// SIMATIC STEP 7 (V5.x) project PROJECT-ETHERNET_en
// CPU: CPU 414-2 DP(1)
// CPU: CPU 414-2 DP(1)
// CPU: CPU 414-2 DP(1)
// station: P_ADR_BUS
// station: Hardware
// station: SIMATIC 400(3)
// station: P_ADR_BUS
// station: Hardware
// station: SIMATIC 400(2)
// station: P_ADR_BUS
// station: Hardware
// station: SIMATIC 400(1)
// program: S7 Program(1)
// program: S7 Program(1)
// program: S7 Program(1)

SYMBOL_TABLE
"AG_SEND"	FC 5	FC 5	// AG SEND
"AG_RECV"	FC 6	FC 6	// AG RECEIVE
END_SYMBOL_TABLE

// FC 5: know-how protected block, not included

// FC 6: know-how protected block, not included

FUNCTION FC 29 : VOID
VERSION : 0.1
BEGIN
NETWORK
TITLE =
      A     T 4;	//time downwards
      JC    runt;
st_1: A     M 40.1;	//start timer 3
      L     S5T#3S;	//LED upwards 3 sec
      SE    T 3;
      A     T 3;
      R     M 40.1;
      JC    hoch;	//jump for upwards
      AN    T 3;
      S     M 40.1;
      S     M 40.2;
runt: A     M 40.2;	//start timer 4
      L     S5T#3S;	//LED downwards 3 sec
      SE    T 4;
      A     T 4;
      R     M 40.2;
      AN    T 4;
      S     M 40.2;
      JC    st_1;
      A     M 40.0;
      L     S5T#100MS;
      SE    T 1;
      A     T 1;
      R     M 40.0;
      A     T 1;
      JC    weit;
      AN    T 1;
      S     M 40.0;
      L     MW 70;
      L     0;
      <>D;
      JC    los1;
      TAK;
      +     1;
      T     MW 70;
      T     DB30.DBW 1;
      BEU;
los1: L     MW 70;
      L     2;
      *D;
      T     MW 70;
      T     DB30.DBW 1;
      L     L#32768;
      <>D;
      BEC;
      L     0;
      T     MW 70;
weit: BEU;
hoch: A     M 40.3;
      L     S5T#100MS;
      SE    T 1;
      A     T 1;
      R     M 40.3;
      A     T 1;
      JC    weit;
      AN    T 1;
      S     M 40.3;
      L     MW 70;
      L     0;
      <>D;
      JC    los2;
      TAK;
      +     L#32768;
      T     MW 70;
      T     DB30.DBW 1;
      BEU;
los2: L     MW 70;
      L     2;
      /D;
      T     MW 70;
      T     DB30.DBW 1;
      L     1;
      <>D;
      BEC;
      L     0;
      T     MW 70;
      BE;
END_FUNCTION

FUNCTION FC 30 : VOID
TITLE = send
//SIMATIC 400 Station 1
//
//Sends data via ISO transport connection with ID=1.
//Starting at byte 1 in DB30, 4 bytes are going to be send.
//
VERSION : 0.0
BEGIN
NETWORK
TITLE =
      O     M 50.0;
      ON    M 50.0;
      S     M 50.0;
      CALL  "AG_SEND" (
           $1                       := P#M 50.0,
           $2                       := 1,
           $3                       := 512,
           $4                       := P#DB30.DBX 1.0 BYTE 240,
           $5                       := 4,
           $6                       := M 1.2,
           $7                       := M 1.3,
           $8                       := P#M 200.0);	//AG_SEND
      BE;
END_FUNCTION

FUNCTION FC 31 : VOID
TITLE = receive
//SIMATIC 400 Station 1
//
//Receives data via ISO transport connection with ID=1.
//Data are accepted in DB31, starting at byte 1.
VERSION : 0.0
BEGIN
NETWORK
TITLE =
      CALL  "AG_RECV" (
           $1                       := 1,
           $2                       := 512,
           $3                       := P#DB31.DBX 1.0 BYTE 240,
           $4                       := P#M 1.0,
           $5                       := M 1.1,
           $6                       := P#M 202.0,
           $7                       := P#M 10.0);	//AG_RECV
      L     DB31.DBW 1;
      T     QW 0;
      BE;
END_FUNCTION

ORGANIZATION_BLOCK OB 1
//Station 1
VERSION : 0.1
VAR_TEMP
  OB1_EV_CLASS : BYTE ;	//Bits 0-3 = 1 (Coming event), Bits 4-7 = 1 (Event class 1)
  OB1_SCAN_1 : BYTE ;	//1 (Cold restart scan 1 of OB 1), 3 (Scan 2-n of OB 1)
  OB1_PRIORITY : BYTE ;	//1 (Priority of 1 is lowest)
  OB1_OB_NUMBR : BYTE ;	//1 (Organization block 1, OB1)
  OB1_RESERVED_1 : BYTE ;	//Reserved for system
  OB1_RESERVED_2 : BYTE ;	//Reserved for system
  OB1_PREV_CYCLE : INT ;	//Cycle time of previous OB1 scan (milliseconds)
  OB1_MIN_CYCLE : INT ;	//Minimum cycle time of OB1 (milliseconds)
  OB1_MAX_CYCLE : INT ;	//Maximum cycle time of OB1 (milliseconds)
  OB1_DATE_TIME : DATE_AND_TIME ;	//Date and time OB1 started
END_VAR
BEGIN
NETWORK
TITLE =
      CALL  FC 29;
      CALL  FC 30;
      CALL  FC 31;
      BE;
END_ORGANIZATION_BLOCK

ORGANIZATION_BLOCK OB 100
TITLE = Start up
//Station1
VERSION : 0.0
VAR_TEMP
  OB100_EV_CLASS : BYTE ;	//16#13, Event class 1, Entering event state, Event logged in diagnostic buffer
  OB100_STRTUP : BYTE ;	//16#81/82/83/84 Method of startup
  OB100_PRIORITY : BYTE ;	//27 (Priority of 1 is lowest)
  OB100_OB_NUMBR : BYTE ;	//100 (Organization block 100, OB100)
  OB100_RESERVED_1 : BYTE ;	//Reserved for system
  OB100_RESERVED_2 : BYTE ;	//Reserved for system
  OB100_STOP : WORD ;	//Event that caused CPU to stop (16#4xxx)
  OB100_STRT_INFO : DWORD ;	//Information on how system started
  OB100_DATE_TIME : DATE_AND_TIME ;	//Date and time OB100 started
END_VAR
BEGIN
NETWORK
TITLE =
//Creation of DB30 and DB31, each with a length about 350 byte
      L     30;
      T     MW 22;
      L     31;
      T     MW 24;
      L     350;
      T     MW 26;
      CALL  SFC 22 (
           LOW_LIMIT                := MW 22,
           UP_LIMIT                 := MW 24,
           COUNT                    := MW 26,
           RET_VAL                  := MW 28,
           DB_NUMBER                := MW 30);
      CALL  SFC 22 (
           LOW_LIMIT                := MW 22,
           UP_LIMIT                 := MW 24,
           COUNT                    := MW 26,
           RET_VAL                  := MW 28,
           DB_NUMBER                := MW 30);
      BE;
END_ORGANIZATION_BLOCK

// FC 5: know-how protected block, not included

// FC 6: know-how protected block, not included

FUNCTION FC 30 : VOID
TITLE = send
//SIMATIC 400 Station 2
//
//Return the data as job confirmation.
VERSION : 0.0
BEGIN
NETWORK
TITLE =
      O     M 50.0;
      ON    M 50.0;
      S     M 50.0;
      CALL  "AG_SEND" (
           $1                       := P#M 50.0,
           $2                       := 1,
           $3                       := 512,
           $4                       := P#DB31.DBX 1.0 BYTE 240,
           $5                       := 4,
           $6                       := M 1.2,
           $7                       := M 1.3,
           $8                       := P#M 200.0);	//AG_SEND
      BE;
END_FUNCTION

FUNCTION FC 31 : VOID
TITLE = receive
//SIMATIC 400 Station 2
//
//Save the received data in the data block and output the data to the process 
//simulation.
VERSION : 0.0
BEGIN
NETWORK
TITLE =
      CALL  "AG_RECV" (
           $1                       := 1,
           $2                       := 512,
           $3                       := P#DB31.DBX 1.0 BYTE 240,
           $4                       := P#M 1.0,
           $5                       := M 1.1,
           $6                       := P#M 202.0,
           $7                       := P#M 10.0);
      L     DB31.DBW 1;
      T     QW 0;
      BE;
END_FUNCTION

ORGANIZATION_BLOCK OB 1
//Station 2
VERSION : 0.1
VAR_TEMP
  OB1_EV_CLASS : BYTE ;	//Bits 0-3 = 1 (Coming event), Bits 4-7 = 1 (Event class 1)
  OB1_SCAN_1 : BYTE ;	//1 (Cold restart scan 1 of OB 1), 3 (Scan 2-n of OB 1)
  OB1_PRIORITY : BYTE ;	//1 (Priority of 1 is lowest)
  OB1_OB_NUMBR : BYTE ;	//1 (Organization block 1, OB1)
  OB1_RESERVED_1 : BYTE ;	//Reserved for system
  OB1_RESERVED_2 : BYTE ;	//Reserved for system
  OB1_PREV_CYCLE : INT ;	//Cycle time of previous OB1 scan (milliseconds)
  OB1_MIN_CYCLE : INT ;	//Minimum cycle time of OB1 (milliseconds)
  OB1_MAX_CYCLE : INT ;	//Maximum cycle time of OB1 (milliseconds)
  OB1_DATE_TIME : DATE_AND_TIME ;	//Date and time OB1 started
END_VAR
BEGIN
NETWORK
TITLE =
      CALL  FC 30;
      CALL  FC 31;
      BE;
END_ORGANIZATION_BLOCK

ORGANIZATION_BLOCK OB 100
TITLE = Station 2
VERSION : 0.0
VAR_TEMP
  OB100_EV_CLASS : BYTE ;	//16#13, Event class 1, Entering event state, Event logged in diagnostic buffer
  OB100_STRTUP : BYTE ;	//16#81/82/83/84 Method of startup
  OB100_PRIORITY : BYTE ;	//27 (Priority of 1 is lowest)
  OB100_OB_NUMBR : BYTE ;	//100 (Organization block 100, OB100)
  OB100_RESERVED_1 : BYTE ;	//Reserved for system
  OB100_RESERVED_2 : BYTE ;	//Reserved for system
  OB100_STOP : WORD ;	//Event that caused CPU to stop (16#4xxx)
  OB100_STRT_INFO : DWORD ;	//Information on how system started
  OB100_DATE_TIME : DATE_AND_TIME ;	//Date and time OB100 started
END_VAR
BEGIN
NETWORK
TITLE =
//Creation of DB30 and DB31, each with a length about 350 byte
      L     30;
      T     MW 22;
      L     31;
      T     MW 24;
      L     250;
      T     MW 26;
      CALL  SFC 22 (
           LOW_LIMIT                := MW 22,
           UP_LIMIT                 := MW 24,
           COUNT                    := MW 26,
           RET_VAL                  := MW 28,
           DB_NUMBER                := MW 30);
      CALL  SFC 22 (
           LOW_LIMIT                := MW 22,
           UP_LIMIT                 := MW 24,
           COUNT                    := MW 26,
           RET_VAL                  := MW 28,
           DB_NUMBER                := MW 30);
      BE;
END_ORGANIZATION_BLOCK

// FC 5: know-how protected block, not included

// FC 6: know-how protected block, not included

FUNCTION FC 29 : VOID
TITLE = handle process data
//SIMATIC 400 Station 3
//
//A data word is incremented and decremented cyclically. The time interval for 
//incrementing and decrementing is 3 seconds.
VERSION : 0.1
BEGIN
NETWORK
TITLE =
      A     T 4;	//Time downwards
      JC    runt;
st_1: A     M 40.1;	//start timer 3
      L     S5T#3S;	//LED upwards 3 sec
      SE    T 3;
      A     T 3;
      R     M 40.1;
      JC    hoch;	//jump for upwards
      AN    T 3;
      S     M 40.1;
      S     M 40.2;
runt: A     M 40.2;	//start timer 4
      L     S5T#3S;	//LED downwards 3 sec
      SE    T 4;
      A     T 4;
      R     M 40.2;
      AN    T 4;
      S     M 40.2;
      JC    st_1;
      A     M 40.0;
      L     S5T#100MS;
      SE    T 1;
      A     T 1;
      R     M 40.0;
      A     T 1;
      JC    weit;
      AN    T 1;
      S     M 40.0;
      L     MW 70;
      L     0;
      <>D;
      JC    los1;
      TAK;
      +     1;
      T     MW 70;
      T     DB30.DBW 1;
      BEU;
los1: L     MW 70;
      L     2;
      *D;
      T     MW 70;
      T     DB30.DBW 1;
      L     L#32768;
      <>D;
      BEC;
      L     0;
      T     MW 70;
weit: BEU;
hoch: A     M 40.3;
      L     S5T#100MS;
      SE    T 1;
      A     T 1;
      R     M 40.3;
      A     T 1;
      JC    weit;
      AN    T 1;
      S     M 40.3;
      L     MW 70;
      L     0;
      <>D;
      JC    los2;
      TAK;
      +     L#32768;
      T     MW 70;
      T     DB30.DBW 1;
      BEU;
los2: L     MW 70;
      L     2;
      /D;
      T     MW 70;
      T     DB30.DBW 1;
      L     1;
      <>D;
      BEC;
      L     0;
      T     MW 70;
      BE;
END_FUNCTION

FUNCTION FC 30 : VOID
TITLE = Senden / send
//SIMATIC 400 Station 3
//
//Sends data via ISO transport connection with ID=1.
//Starting at byte 1 in DB30, 4 bytes are going to be send.
VERSION : 0.0
BEGIN
NETWORK
TITLE =
      O     M 50.0;
      ON    M 50.0;
      S     M 50.0;
      CALL  "AG_SEND" (
           $1                       := P#M 50.0,
           $2                       := 1,
           $3                       := 512,
           $4                       := P#DB30.DBX 1.0 BYTE 240,
           $5                       := 4,
           $6                       := M 1.2,
           $7                       := M 1.3,
           $8                       := P#M 200.0);	//send to S5
      BE;
END_FUNCTION

ORGANIZATION_BLOCK OB 1
VERSION : 0.1
VAR_TEMP
  OB1_EV_CLASS : BYTE ;	//Bits 0-3 = 1 (Coming event), Bits 4-7 = 1 (Event class 1)
  OB1_SCAN_1 : BYTE ;	//1 (Cold restart scan 1 of OB 1), 3 (Scan 2-n of OB 1)
  OB1_PRIORITY : BYTE ;	//1 (Priority of 1 is lowest)
  OB1_OB_NUMBR : BYTE ;	//1 (Organization block 1, OB1)
  OB1_RESERVED_1 : BYTE ;	//Reserved for system
  OB1_RESERVED_2 : BYTE ;	//Reserved for system
  OB1_PREV_CYCLE : INT ;	//Cycle time of previous OB1 scan (milliseconds)
  OB1_MIN_CYCLE : INT ;	//Minimum cycle time of OB1 (milliseconds)
  OB1_MAX_CYCLE : INT ;	//Maximum cycle time of OB1 (milliseconds)
  OB1_DATE_TIME : DATE_AND_TIME ;	//Date and time OB1 started
END_VAR
BEGIN
NETWORK
TITLE =
      CALL  FC 29;
      CALL  FC 30;
      BE;
END_ORGANIZATION_BLOCK

ORGANIZATION_BLOCK OB 100
TITLE = Anlauf
//Station1
VERSION : 0.0
VAR_TEMP
  OB100_EV_CLASS : BYTE ;	//16#13, Event class 1, Entering event state, Event logged in diagnostic buffer
  OB100_STRTUP : BYTE ;	//16#81/82/83/84 Method of startup
  OB100_PRIORITY : BYTE ;	//27 (Priority of 1 is lowest)
  OB100_OB_NUMBR : BYTE ;	//100 (Organization block 100, OB100)
  OB100_RESERVED_1 : BYTE ;	//Reserved for system
  OB100_RESERVED_2 : BYTE ;	//Reserved for system
  OB100_STOP : WORD ;	//Event that caused CPU to stop (16#4xxx)
  OB100_STRT_INFO : DWORD ;	//Information on how system started
  OB100_DATE_TIME : DATE_AND_TIME ;	//Date and time OB100 started
END_VAR
BEGIN
NETWORK
TITLE =
//Creation of DB30 and DB31, each with a length about 350 byte
      L     30;
      T     MW 22;
      L     31;
      T     MW 24;
      L     350;
      T     MW 26;
      CALL  SFC 22 (
           LOW_LIMIT                := MW 22,
           UP_LIMIT                 := MW 24,
           COUNT                    := MW 26,
           RET_VAL                  := MW 28,
           DB_NUMBER                := MW 30);
      CALL  SFC 22 (
           LOW_LIMIT                := MW 22,
           UP_LIMIT                 := MW 24,
           COUNT                    := MW 26,
           RET_VAL                  := MW 28,
           DB_NUMBER                := MW 30);
      BE;
END_ORGANIZATION_BLOCK
